FUNCTION_BLOCK fb_CreateTable
VAR_INPUT
	tablename:STRING(50);
END_VAR
VAR_OUTPUT
	bReady:BOOL:=FALSE;
END_VAR
VAR
	bExecute:Bool:=false;
END_VAR

METHOD execute : BOOL
VAR_INPUT
END_VAR
bExecute:=TRUE;
END_METHOD

METHOD reset : BOOL
VAR_INPUT
END_VAR
bExecute:=FALSE;
bReady:=false;
END_METHOD

END_FUNCTION_BLOCK

(* stored: Version 1.1.0.1, ProductVersion 3.1.4024.2
   POU fb_CreateTable: Id {d3fe11d2-ae59-4531-b2d9-57fd37adc6ac}, SpecialFunc None
   Method execute: Id {ec82c688-b6d3-4299-bfec-664a40218274}
   Method reset: Id {faa612af-0d76-4df4-984d-7446ad233771} *)
